TYPE "SinamicsCU_Alarms"
VERSION : 0.1
// Block: SinamicsCU_Alarms
   STRUCT
      CUFault : Bool;
      CommunicationFault : Bool;
   END_STRUCT;

END_TYPE
